// TIA Portal V20 export
DATA_BLOCK "ShiftInitBools"   // DB257
// stored: MemoryReserve 100
   VAR
      earlyShift : Bool := FALSE;
      lateShift : Bool := FALSE;
      nightShift : Bool := FALSE;
   END_VAR
BEGIN
END_DATA_BLOCK
